Staubli VAL3: ListMsg.pgx

program ListMsg(bool x_bRefresh (dimensions=1), string x_sS (dimensions=1))
begin
  switch sLanguge
    case "English"
      call ListMsgE(x_bRefresh,x_sS)
    break
    case "Chinese"
      call ListMsgC(x_bRefresh,x_sS)
    break
  endSwitch
end
